FUNCTION_BLOCK ILOCK_CONFLICT_TRIP (* Prioritizes the first active input and trips on conflict. Requires RESET. *)
  (* Standard: 61499-2; Description: Copyright (c) 2023 HR Agrartechnik GmbH This program and the accompanying materials are made available under the terms of the Eclipse Public License 2.0 which is available at https://www.eclipse.org/legal/epl-2.0/ SPDX-License-Identifier: EPL-2.0 *)
  (* Version 1.0, 2026-04-19, Franz Höpfinger, HR Agrartechnik GmbH, initial API and implementation and/or initial documentation *)
  PACKAGE logiBUS::signalprocessing::interlock;
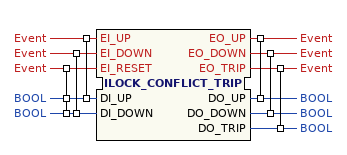
  EVENT_INPUT
    EI_UP WITH DI_UP;
    EI_DOWN WITH DI_DOWN;
    EI_RESET WITH DI_UP, DI_DOWN;
  END_EVENT
  EVENT_OUTPUT
    EO_UP WITH DO_UP;
    EO_DOWN WITH DO_DOWN;
    EO_TRIP WITH DO_TRIP;
  END_EVENT
  VAR_INPUT
    DI_UP : BOOL; (* TRUE = forward, up, right, clockwise *)
    DI_DOWN : BOOL; (* TRUE = backward, down, left, counter-clockwise *)
  END_VAR
  VAR_OUTPUT
    DO_UP : BOOL; (* TRUE = forward, up, right, clockwise *)
    DO_DOWN : BOOL; (* TRUE = backward, down, left, counter-clockwise *)
    DO_TRIP : BOOL; (* TRUE = Conflict/Trip state active *)
  END_VAR
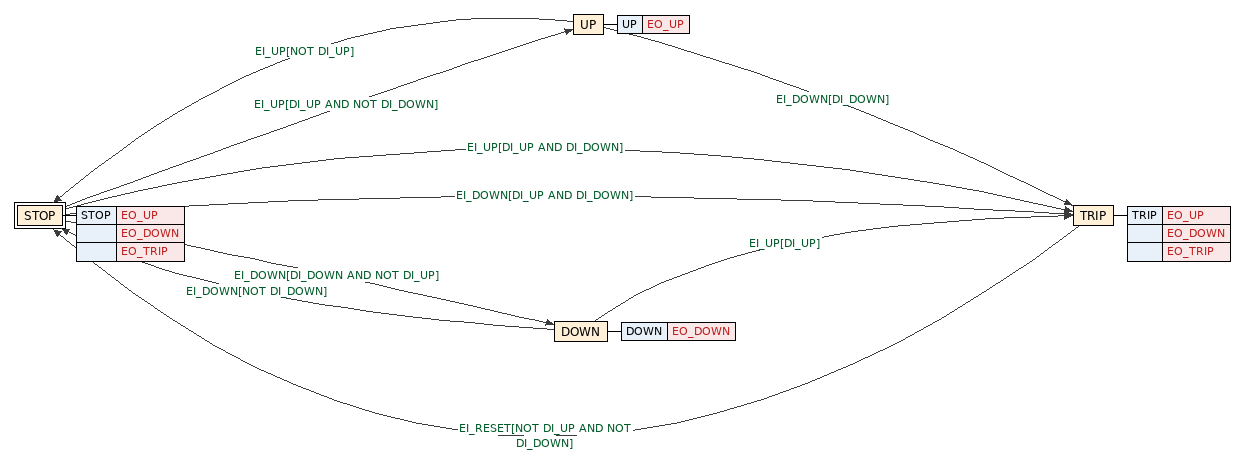
  EC_STATES
    STOP : STOP -> EO_UP, -> EO_DOWN, -> EO_TRIP;
    UP : UP -> EO_UP;
    DOWN : DOWN -> EO_DOWN;
    TRIP : TRIP -> EO_UP, -> EO_DOWN, -> EO_TRIP;
  END_STATES
  EC_TRANSITIONS
    STOP TO UP := EI_UP[DI_UP AND NOT DI_DOWN];
    STOP TO DOWN := EI_DOWN[DI_DOWN AND NOT DI_UP];
    STOP TO TRIP := EI_UP[DI_UP AND DI_DOWN];
    STOP TO TRIP := EI_DOWN[DI_UP AND DI_DOWN];
    UP TO STOP := EI_UP[NOT DI_UP];
    UP TO TRIP := EI_DOWN[DI_DOWN];
    DOWN TO STOP := EI_DOWN[NOT DI_DOWN];
    DOWN TO TRIP := EI_UP[DI_UP];
    TRIP TO STOP := EI_RESET[NOT DI_UP AND NOT DI_DOWN];
  END_TRANSITIONS
  ALGORITHM UP IN ST:
DO_UP := BOOL#TRUE;
DO_DOWN := BOOL#FALSE;
DO_TRIP := BOOL#FALSE;
  END_ALGORITHM
  ALGORITHM DOWN IN ST:
DO_UP := BOOL#FALSE;
DO_DOWN := BOOL#TRUE;
DO_TRIP := BOOL#FALSE;
  END_ALGORITHM
  ALGORITHM STOP IN ST:
DO_UP := BOOL#FALSE;
DO_DOWN := BOOL#FALSE;
DO_TRIP := BOOL#FALSE;
  END_ALGORITHM
  ALGORITHM TRIP IN ST:
DO_UP := BOOL#FALSE;
DO_DOWN := BOOL#FALSE;
DO_TRIP := BOOL#TRUE;
  END_ALGORITHM
END_FUNCTION_BLOCK
